{attribute 'qualified_only'}
VAR_GLOBAL CONSTANT
	nMAX_MESSAGES_SHOWN 	: UDINT := 10 	;
	nMAX_MESSAGE_HISTORY	: UDINT := 1000 ;
	nMAX_CSV_FIELD_LENGTH	: UDINT := 100	;
	tMESSAGE_TIMEOUT		: TIME 	:= T#10S ;
	sLOGFILE_PATH			: STRING:= 'D:\FaultLogs\'	;
	sLOGFILE_NAME			: STRING:= 'Faultlog' 		; // Message log destination file
	nMESSAGE_COLUMNS		: UDINT := 8 ;
	tOMCYCLETIME			: TIME 	:= T#5S  ; // Time that an operator message is shown before it cycles to the next OM
END_VAR

(* stored: Version 1.1.0.1, ProductVersion 3.1.4024.10
   GVL Param_Messages: Id {2016c387-f096-4466-aaa3-690b7ef65799}, ParameterList True *)
